// TIA Portal V21 export
VAR_GLOBAL   // PLC tag table "BIT"
END_VAR
